// TwinCAT 3 PLC project LogicEffectOnIOReliability
// ProgramVersion: 3.1.4020.4
// libraries:
//   Tc2_Standard, * (Beckhoff Automation GmbH)
//   Tc2_System, * (Beckhoff Automation GmbH)
//   Tc3_Module, * (Beckhoff Automation GmbH)
// project tree:
//   DUTs/ DigitalInput.TcDUT, DigitalOutput.TcDUT
//   / PlcTask.TcTTO
//   POUs/ iterator.TcPOU, MAIN.TcPOU

CONFIGURATION LogicEffectOnIOReliability
    RESOURCE PLC ON TwinCAT3
        TASK PlcTask(INTERVAL := T#50us, PRIORITY := 20);
        PROGRAM MAIN WITH PlcTask : MAIN;
    END_RESOURCE
END_CONFIGURATION

// ---- DUTs/DigitalInput.TcDUT
TYPE DigitalInput :
STRUCT
	in AT %I*	:	BIT;
END_STRUCT
END_TYPE

// ---- DUTs/DigitalOutput.TcDUT
TYPE DigitalOutput :
STRUCT
	out AT %Q*	:	BIT;
END_STRUCT
END_TYPE

// ---- POUs/MAIN.TcPOU
PROGRAM MAIN
VAR
	// CPU Manipulator
	itr_enb	:	BOOL	:=	TRUE;
	cpu_enb	:	BOOL	:=	TRUE;
	ulimit	:	DINT	:=	1000;
	delay	:	DINT	:=	50;
	assign	:	BOOL	:=	FALSE;
	(**********************)
	arr	:	ARRAY	[0..20000]	OF	iterator;
	cache	:	ARRAY	[0..20000]	OF	DINT;
	noToTest	:	DINT	:= 0;
	count	: DINT	:=0;
	I	:	DINT;
	step	:	BOOL;
	
	// IO operator
	io_enb	:	BOOL	:=	TRUE;
	starter	:	DigitalOutput;
	input	:	DigitalInput;
	output	:	DigitalOutput;
	term	:	DigitalInput;
	counter	:	UINT	:=	0;
	c_limit	:	UINT 	:= 100;
	s_limit	:	UINT	:=90;
END_VAR

// CPU manipulator
IF itr_enb THEN
	IF count < delay-1 THEN
		count := count + 1;
		step :=	FALSE;
	ELSE
		count := 0;
		step :=	TRUE;
	END_IF
	
	IF step THEN
		IF noToTest < ulimit-1 THEN
			noToTest := noToTest + 1;
		ELSE
			noToTest := 0;
		END_IF
	END_IF
END_IF

IF cpu_enb THEN
	// Run noToTest operations
	FOR I:=0 TO noToTest BY 1 DO 
		arr[I](increment:=1);
		IF ASSIGN THEN
			cache[I] := arr[i].out;
		END_IF
	END_FOR;
END_IF

IF io_enb THEN
	IF counter < c_limit THEN
		counter := counter + 1;
	ELSIF counter >= c_limit THEN
		counter := 0;
	END_IF;
	
	IF counter > s_limit THEN
		starter.out := 1;
	ELSE
		starter.out := 0;
	END_IF
	
	IF input.in THEN
		output.out := 1;
	ELSE
		output.out := 0;
	END_IF
END_IF

END_PROGRAM

// ---- POUs/iterator.TcPOU
FUNCTION_BLOCK iterator
VAR_INPUT
	increment	:	DINT;
END_VAR
VAR_OUTPUT
	out	:	DINT;
END_VAR
VAR
	value	:	DINT	:=0;
	lim	:	DINT :=1000;
END_VAR

IF value < lim THEN
	value := value + increment;
ELSE
	value:= 0;	
END_IF
out := value;

END_FUNCTION_BLOCK
